(* Logix 5000 project; controller SX_V040001_C001 vendor 1 type 14 code 77 rev 16.22; software revision 16.04; part 5 of 35 *)
(* tags used below, declared in another part *)
   ALARM_BITS : INT[10];
   ALL_KINDS : INT[90];
   Basic : INT;
   EMPTYING : INT[18];
   G_AInput : DINT[8];
   G_DInput : DINT[3];
   G_DOutput : DINT[3];
   loading : INT[19];
   m_alarm_exist : BOOL;
   m_notstop : BOOL;
   METERING : INT[44];
   PARAMETER : INT[501];
   T_AIR_PRESSURE : TIMER;
   T_BEARING_LUBR : TIMER;
   T_CHOCO_PRESSURE : TIMER;
   T_DELAY_BROKEN_AI_0 : TIMER;
   T_DELAY_BROKEN_AI_1 : TIMER;
   T_DELAY_BROKEN_AI_2 : TIMER;
   T_DELAY_BROKEN_AI_3 : TIMER;
   T_DELAY_BROKEN_AI_4 : TIMER;
   T_DELAY_BROKEN_AI_5 : TIMER;
   T_DELAY_BROKEN_AI_6 : TIMER;
   T_DELAY_BROKEN_AI_7 : TIMER;
   T_INLETT_VALVE : TIMER;
   T_STUFFINGBOX_LUBR : TIMER;
   TEMP : INT[14];
   Z30 : COUNTER;
   Z31 : COUNTER;
   Z33 : COUNTER;
   Z34 : COUNTER;
   Z35 : COUNTER;
   Z36 : COUNTER;
   Z37 : COUNTER;
   Z38 : COUNTER;
   Z39 : COUNTER;
   Z40 : COUNTER;
   Z41 : COUNTER;
(* MainProgram, continued *)

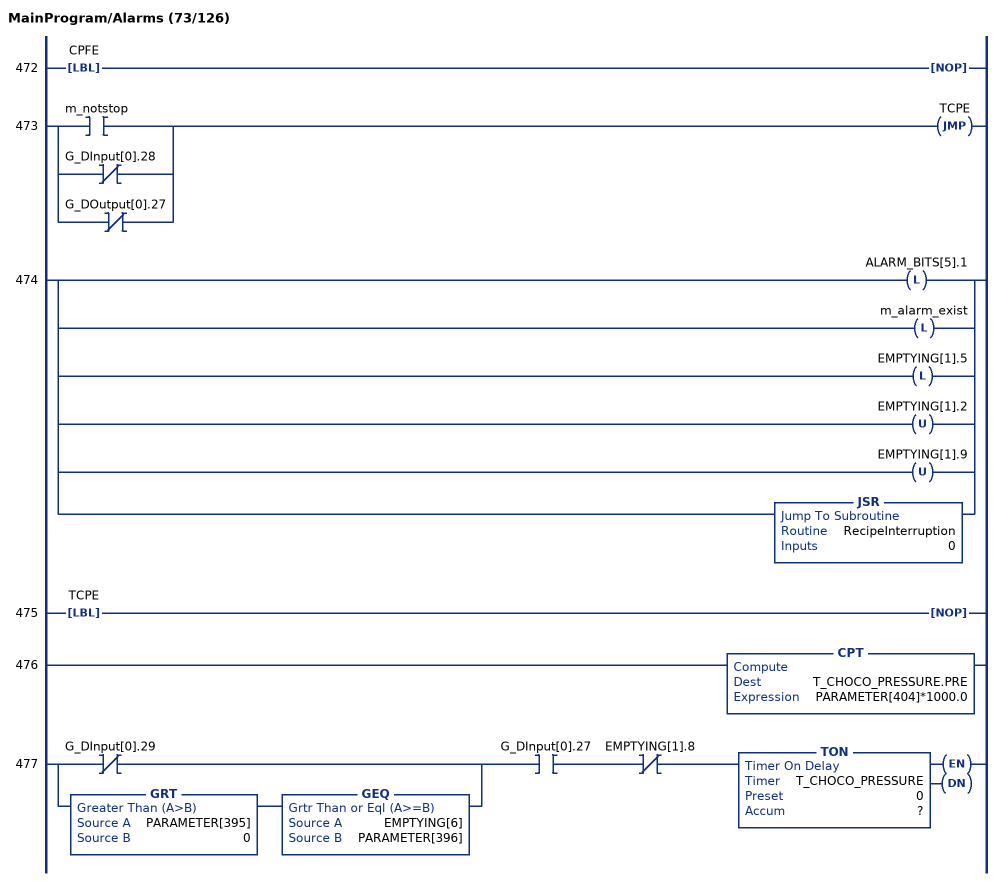
   [picture p94: MainProgram/Alarms rungs 472-477]
   472: LBL(CPFE)NOP();
   473: [XIC(m_notstop) ,XIO(G_DInput[0].28) ,XIO(G_DOutput[0].27) ]JMP(TCPE);
   474: [OTL(ALARM_BITS[5].1) ,OTL(m_alarm_exist) ,OTL(EMPTYING[1].5) ,OTU(EMPTYING[1].2) ,OTU(EMPTYING[1].9) ,JSR(RecipeInterruption,0) ];
   475: LBL(TCPE)NOP();
   476: CPT(T_CHOCO_PRESSURE.PRE,PARAMETER[404]*1000.0);
   477: [XIO(G_DInput[0].29) ,GRT(PARAMETER[395],0) GEQ(EMPTYING[6],PARAMETER[396]) ]XIC(G_DInput[0].27)XIO(EMPTYING[1].8)TON(T_CHOCO_PRESSURE,?,?);
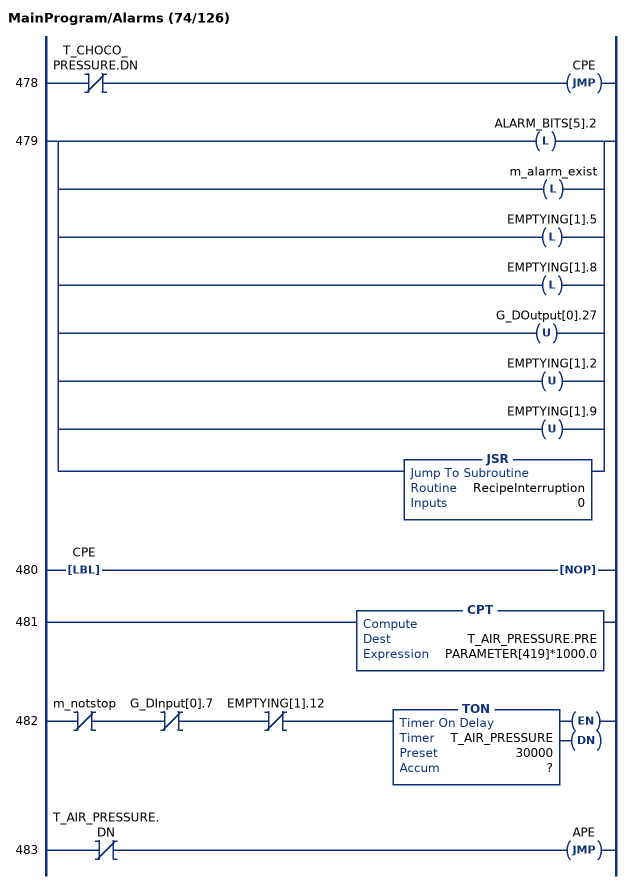
   478: XIO(T_CHOCO_PRESSURE.DN)JMP(CPE);
   479: [OTL(ALARM_BITS[5].2) ,OTL(m_alarm_exist) ,OTL(EMPTYING[1].5) ,OTL(EMPTYING[1].8) ,OTU(G_DOutput[0].27) ,OTU(EMPTYING[1].2) ,OTU(EMPTYING[1].9) ,JSR(RecipeInterruption,0) ];
   480: LBL(CPE)NOP();
   481: CPT(T_AIR_PRESSURE.PRE,PARAMETER[419]*1000.0);
   482: XIO(m_notstop)XIO(G_DInput[0].7)XIO(EMPTYING[1].12)TON(T_AIR_PRESSURE,?,?);
   483: XIO(T_AIR_PRESSURE.DN)JMP(APE);
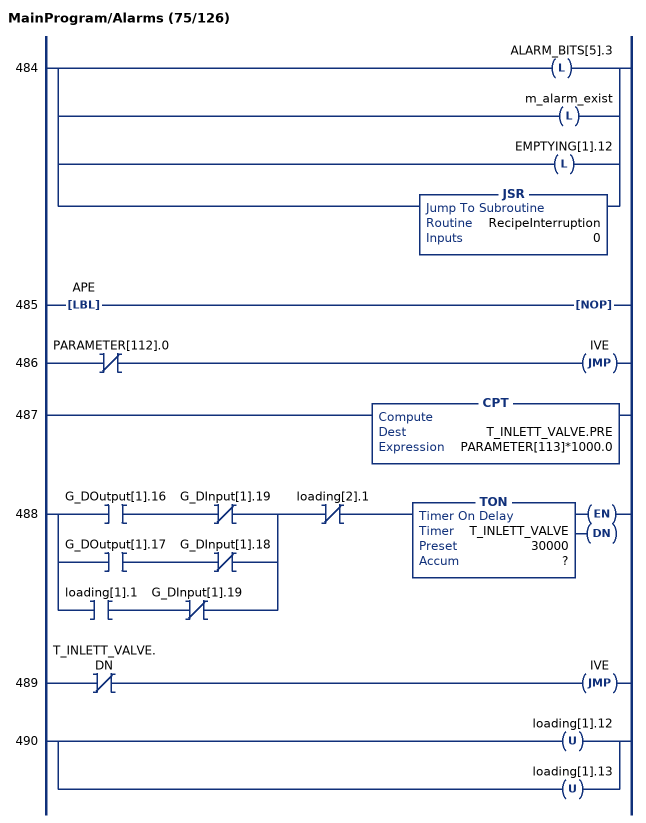
   484: [OTL(ALARM_BITS[5].3) ,OTL(m_alarm_exist) ,OTL(EMPTYING[1].12) ,JSR(RecipeInterruption,0) ];
   485: LBL(APE)NOP();
   486: XIO(PARAMETER[112].0)JMP(IVE);
   487: CPT(T_INLETT_VALVE.PRE,PARAMETER[113]*1000.0);
   488: [XIC(G_DOutput[1].16) XIO(G_DInput[1].19) ,XIC(G_DOutput[1].17) XIO(G_DInput[1].18) ,XIC(loading[1].1) XIO(G_DInput[1].19) ]XIO(loading[2].1)TON(T_INLETT_VALVE,?,?);
   489: XIO(T_INLETT_VALVE.DN)JMP(IVE);
   490: [OTU(loading[1].12) ,OTU(loading[1].13) ];
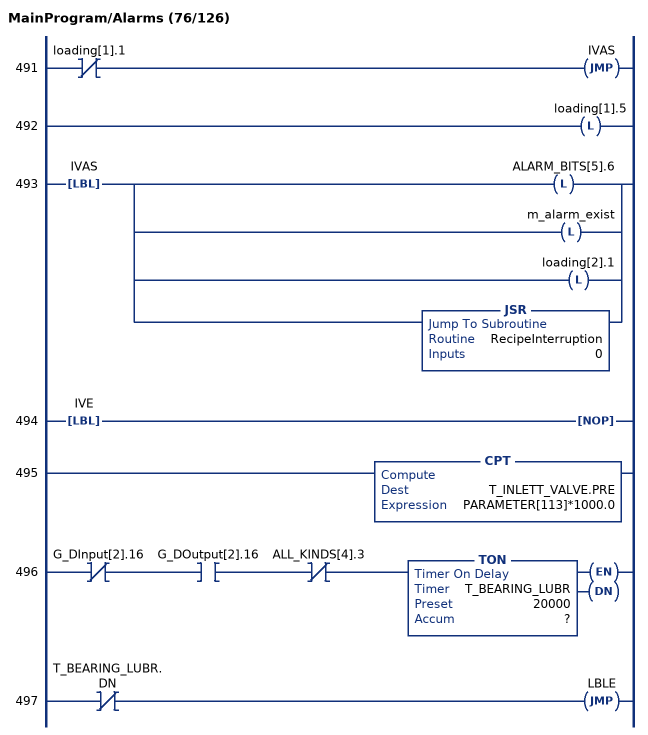
   491: XIO(loading[1].1)JMP(IVAS);
   492: OTL(loading[1].5);
   493: LBL(IVAS)[OTL(ALARM_BITS[5].6) ,OTL(m_alarm_exist) ,OTL(loading[2].1) ,JSR(RecipeInterruption,0) ];
   494: LBL(IVE)NOP();
   495: CPT(T_INLETT_VALVE.PRE,PARAMETER[113]*1000.0);
   496: XIO(G_DInput[2].16)XIC(G_DOutput[2].16)XIO(ALL_KINDS[4].3)TON(T_BEARING_LUBR,?,?);
   497: XIO(T_BEARING_LUBR.DN)JMP(LBLE);
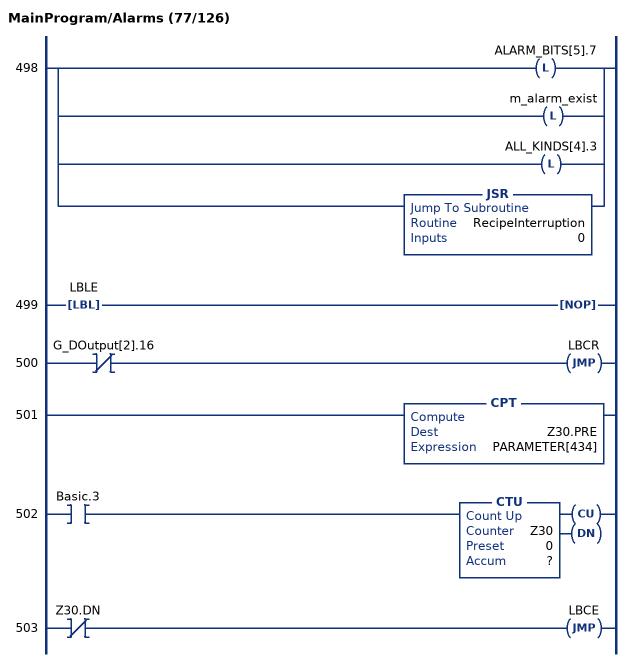
   498: [OTL(ALARM_BITS[5].7) ,OTL(m_alarm_exist) ,OTL(ALL_KINDS[4].3) ,JSR(RecipeInterruption,0) ];
   499: LBL(LBLE)NOP();
   500: XIO(G_DOutput[2].16)JMP(LBCR);
   501: CPT(Z30.PRE,PARAMETER[434]);
   502: XIC(Basic.3)CTU(Z30,?,?);
   503: XIO(Z30.DN)JMP(LBCE);
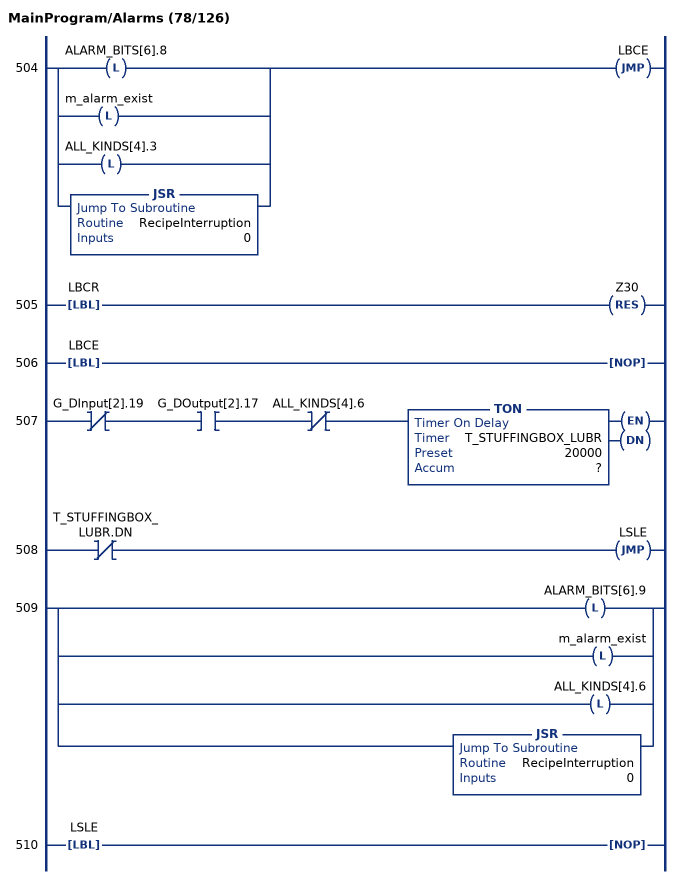
   504: [OTL(ALARM_BITS[6].8) ,OTL(m_alarm_exist) ,OTL(ALL_KINDS[4].3) ,JSR(RecipeInterruption,0) ]JMP(LBCE);
   505: LBL(LBCR)RES(Z30);
   506: LBL(LBCE)NOP();
   507: XIO(G_DInput[2].19)XIC(G_DOutput[2].17)XIO(ALL_KINDS[4].6)TON(T_STUFFINGBOX_LUBR,?,?);
   508: XIO(T_STUFFINGBOX_LUBR.DN)JMP(LSLE);
   509: [OTL(ALARM_BITS[6].9) ,OTL(m_alarm_exist) ,OTL(ALL_KINDS[4].6) ,JSR(RecipeInterruption,0) ];
   510: LBL(LSLE)NOP();
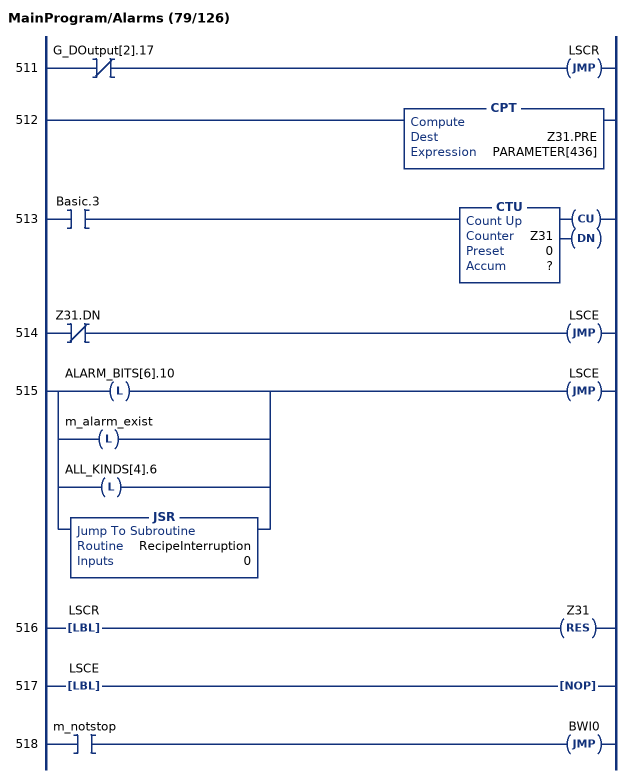
   511: XIO(G_DOutput[2].17)JMP(LSCR);
   512: CPT(Z31.PRE,PARAMETER[436]);
   513: XIC(Basic.3)CTU(Z31,?,?);
   514: XIO(Z31.DN)JMP(LSCE);
   515: [OTL(ALARM_BITS[6].10) ,OTL(m_alarm_exist) ,OTL(ALL_KINDS[4].6) ,JSR(RecipeInterruption,0) ]JMP(LSCE);
   516: LBL(LSCR)RES(Z31);
   517: LBL(LSCE)NOP();
   518: XIC(m_notstop)JMP(BWI0);
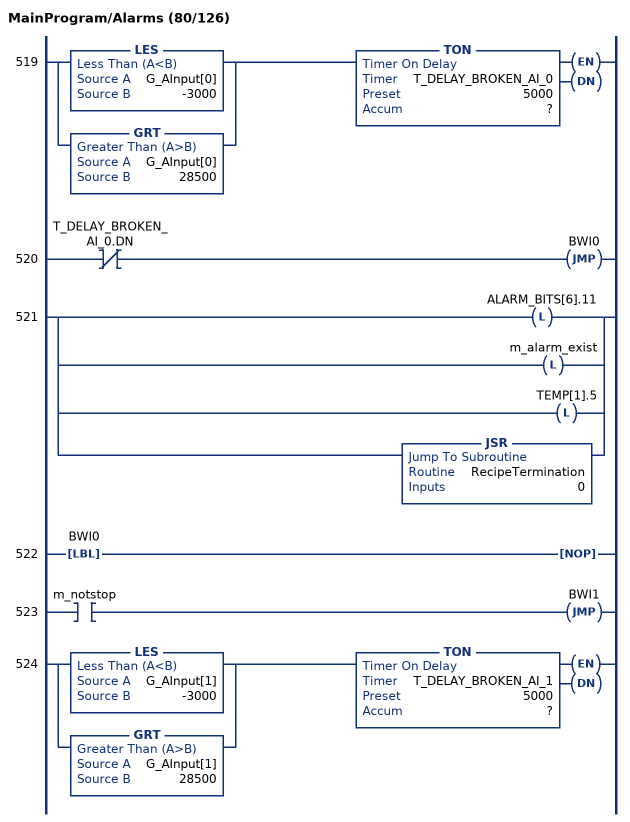
   519: [LES(G_AInput[0],-3000) ,GRT(G_AInput[0],28500) ]TON(T_DELAY_BROKEN_AI_0,?,?);
   520: XIO(T_DELAY_BROKEN_AI_0.DN)JMP(BWI0);
   521: [OTL(ALARM_BITS[6].11) ,OTL(m_alarm_exist) ,OTL(TEMP[1].5) ,JSR(RecipeTermination,0) ];
   522: LBL(BWI0)NOP();
   523: XIC(m_notstop)JMP(BWI1);
   524: [LES(G_AInput[1],-3000) ,GRT(G_AInput[1],28500) ]TON(T_DELAY_BROKEN_AI_1,?,?);
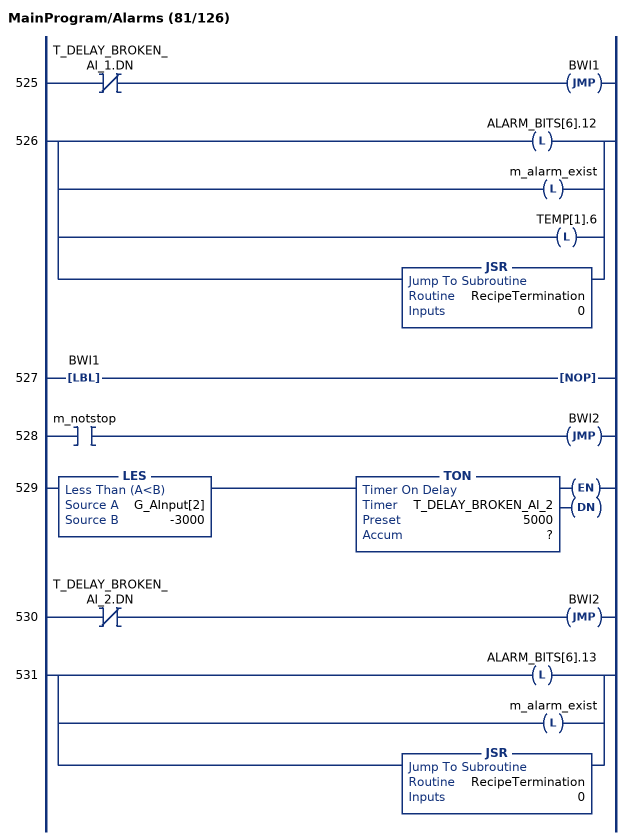
   525: XIO(T_DELAY_BROKEN_AI_1.DN)JMP(BWI1);
   526: [OTL(ALARM_BITS[6].12) ,OTL(m_alarm_exist) ,OTL(TEMP[1].6) ,JSR(RecipeTermination,0) ];
   527: LBL(BWI1)NOP();
   528: XIC(m_notstop)JMP(BWI2);
   529: LES(G_AInput[2],-3000)TON(T_DELAY_BROKEN_AI_2,?,?);
   530: XIO(T_DELAY_BROKEN_AI_2.DN)JMP(BWI2);
   531: [OTL(ALARM_BITS[6].13) ,OTL(m_alarm_exist) ,JSR(RecipeTermination,0) ];
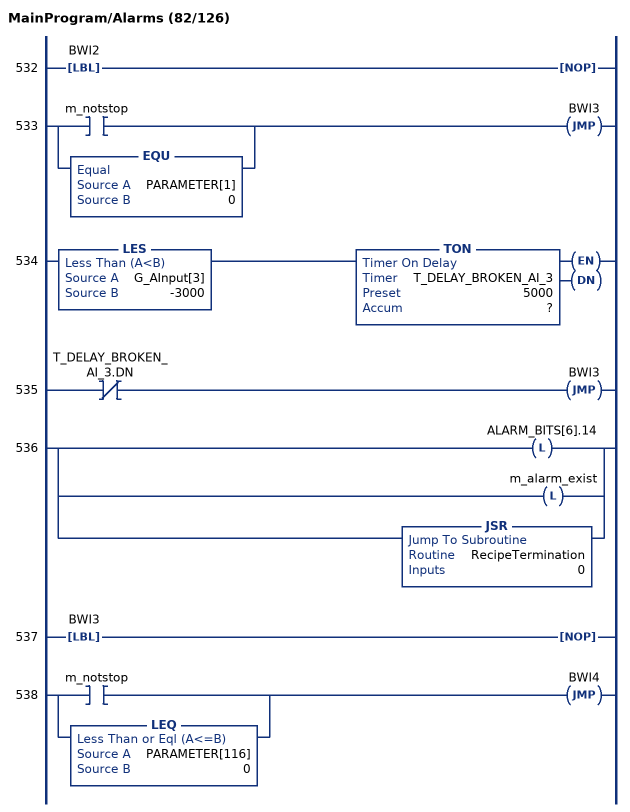
   532: LBL(BWI2)NOP();
   533: [XIC(m_notstop) ,EQU(PARAMETER[1],0) ]JMP(BWI3);
   534: LES(G_AInput[3],-3000)TON(T_DELAY_BROKEN_AI_3,?,?);
   535: XIO(T_DELAY_BROKEN_AI_3.DN)JMP(BWI3);
   536: [OTL(ALARM_BITS[6].14) ,OTL(m_alarm_exist) ,JSR(RecipeTermination,0) ];
   537: LBL(BWI3)NOP();
   538: [XIC(m_notstop) ,LEQ(PARAMETER[116],0) ]JMP(BWI4);
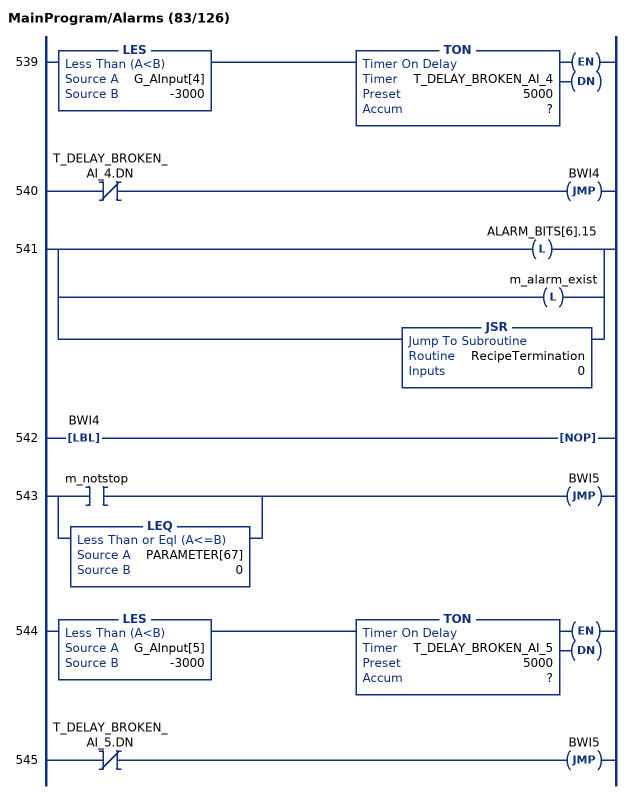
   539: LES(G_AInput[4],-3000)TON(T_DELAY_BROKEN_AI_4,?,?);
   540: XIO(T_DELAY_BROKEN_AI_4.DN)JMP(BWI4);
   541: [OTL(ALARM_BITS[6].15) ,OTL(m_alarm_exist) ,JSR(RecipeTermination,0) ];
   542: LBL(BWI4)NOP();
   543: [XIC(m_notstop) ,LEQ(PARAMETER[67],0) ]JMP(BWI5);
   544: LES(G_AInput[5],-3000)TON(T_DELAY_BROKEN_AI_5,?,?);
   545: XIO(T_DELAY_BROKEN_AI_5.DN)JMP(BWI5);
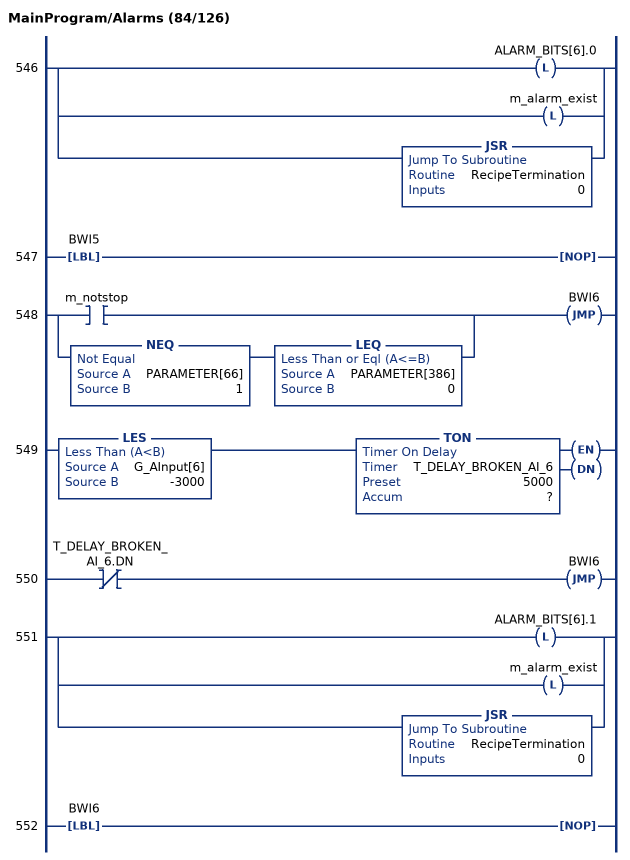
   546: [OTL(ALARM_BITS[6].0) ,OTL(m_alarm_exist) ,JSR(RecipeTermination,0) ];
   547: LBL(BWI5)NOP();
   548: [XIC(m_notstop) ,NEQ(PARAMETER[66],1) LEQ(PARAMETER[386],0) ]JMP(BWI6);
   549: LES(G_AInput[6],-3000)TON(T_DELAY_BROKEN_AI_6,?,?);
   550: XIO(T_DELAY_BROKEN_AI_6.DN)JMP(BWI6);
   551: [OTL(ALARM_BITS[6].1) ,OTL(m_alarm_exist) ,JSR(RecipeTermination,0) ];
   552: LBL(BWI6)NOP();
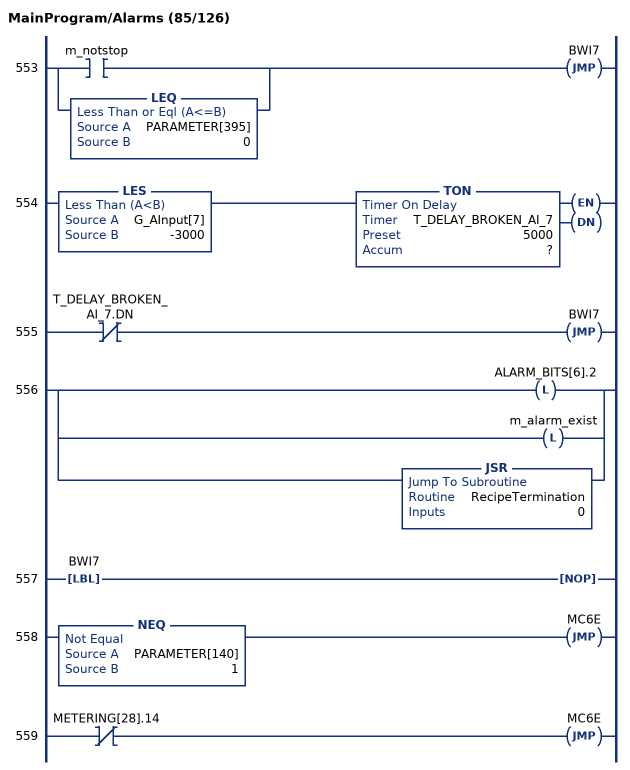
   553: [XIC(m_notstop) ,LEQ(PARAMETER[395],0) ]JMP(BWI7);
   554: LES(G_AInput[7],-3000)TON(T_DELAY_BROKEN_AI_7,?,?);
   555: XIO(T_DELAY_BROKEN_AI_7.DN)JMP(BWI7);
   556: [OTL(ALARM_BITS[6].2) ,OTL(m_alarm_exist) ,JSR(RecipeTermination,0) ];
   557: LBL(BWI7)NOP();
   558: NEQ(PARAMETER[140],1)JMP(MC6E);
   559: XIO(METERING[28].14)JMP(MC6E);
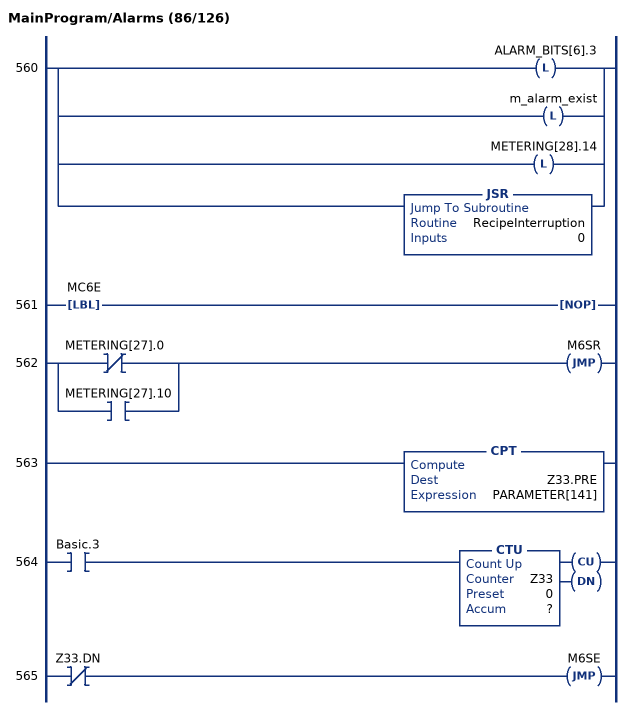
   560: [OTL(ALARM_BITS[6].3) ,OTL(m_alarm_exist) ,OTL(METERING[28].14) ,JSR(RecipeInterruption,0) ];
   561: LBL(MC6E)NOP();
   562: [XIO(METERING[27].0) ,XIC(METERING[27].10) ]JMP(M6SR);
   563: CPT(Z33.PRE,PARAMETER[141]);
   564: XIC(Basic.3)CTU(Z33,?,?);
   565: XIO(Z33.DN)JMP(M6SE);
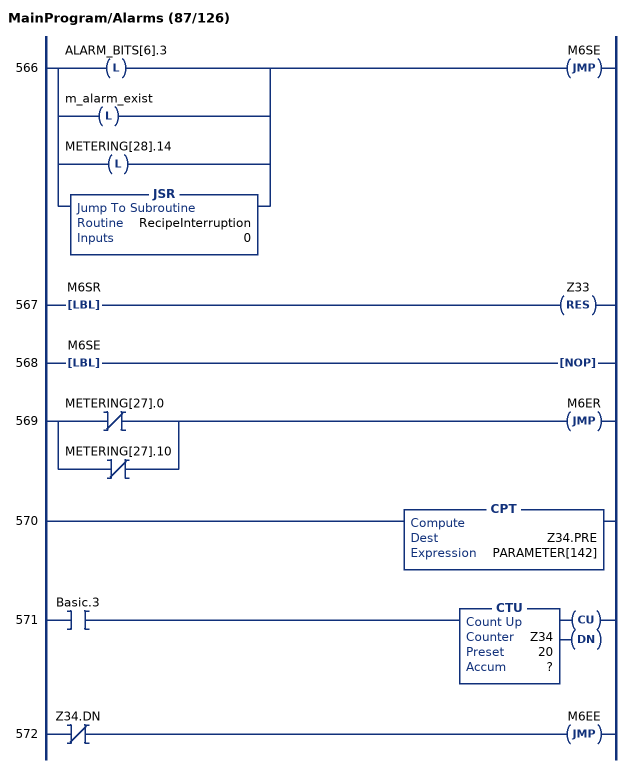
   566: [OTL(ALARM_BITS[6].3) ,OTL(m_alarm_exist) ,OTL(METERING[28].14) ,JSR(RecipeInterruption,0) ]JMP(M6SE);
   567: LBL(M6SR)RES(Z33);
   568: LBL(M6SE)NOP();
   569: [XIO(METERING[27].0) ,XIO(METERING[27].10) ]JMP(M6ER);
   570: CPT(Z34.PRE,PARAMETER[142]);
   571: XIC(Basic.3)CTU(Z34,?,?);
   572: XIO(Z34.DN)JMP(M6EE);
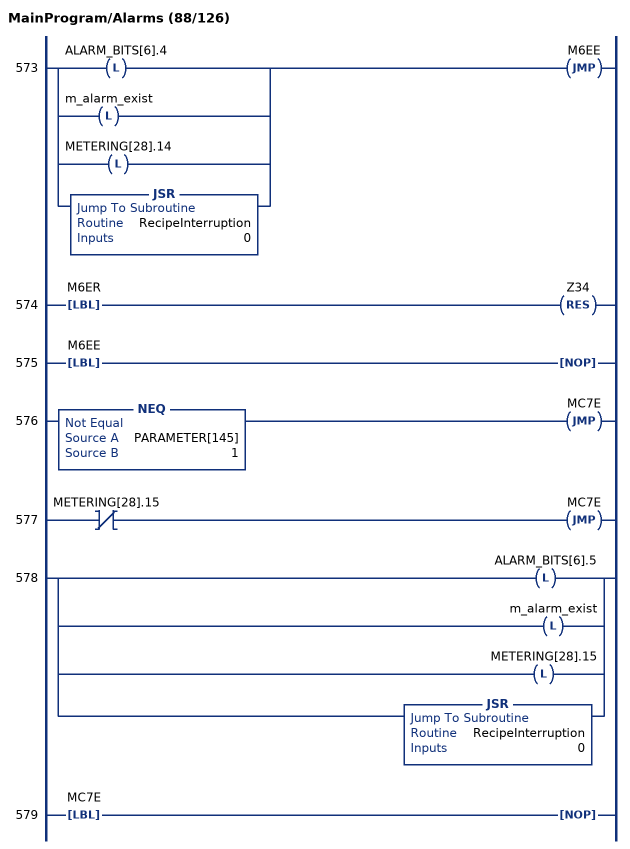
   573: [OTL(ALARM_BITS[6].4) ,OTL(m_alarm_exist) ,OTL(METERING[28].14) ,JSR(RecipeInterruption,0) ]JMP(M6EE);
   574: LBL(M6ER)RES(Z34);
   575: LBL(M6EE)NOP();
   576: NEQ(PARAMETER[145],1)JMP(MC7E);
   577: XIO(METERING[28].15)JMP(MC7E);
   578: [OTL(ALARM_BITS[6].5) ,OTL(m_alarm_exist) ,OTL(METERING[28].15) ,JSR(RecipeInterruption,0) ];
   579: LBL(MC7E)NOP();
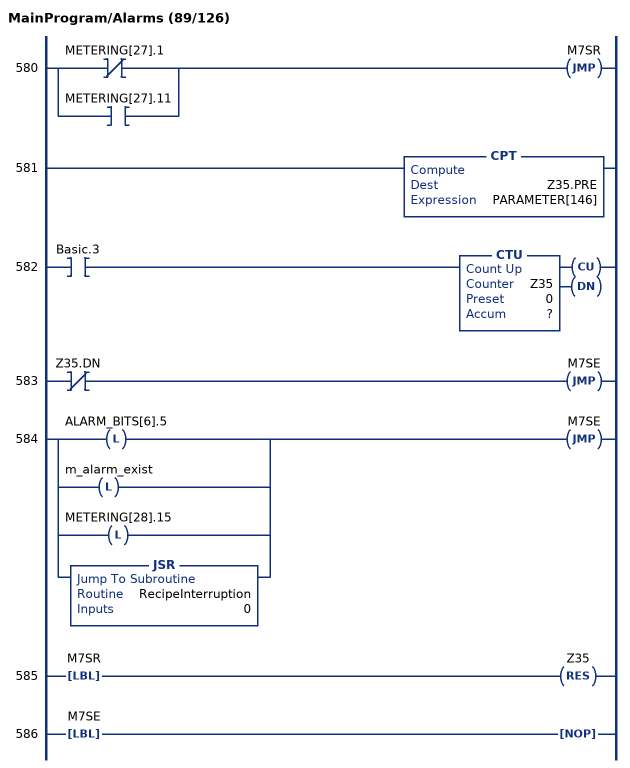
   580: [XIO(METERING[27].1) ,XIC(METERING[27].11) ]JMP(M7SR);
   581: CPT(Z35.PRE,PARAMETER[146]);
   582: XIC(Basic.3)CTU(Z35,?,?);
   583: XIO(Z35.DN)JMP(M7SE);
   584: [OTL(ALARM_BITS[6].5) ,OTL(m_alarm_exist) ,OTL(METERING[28].15) ,JSR(RecipeInterruption,0) ]JMP(M7SE);
   585: LBL(M7SR)RES(Z35);
   586: LBL(M7SE)NOP();
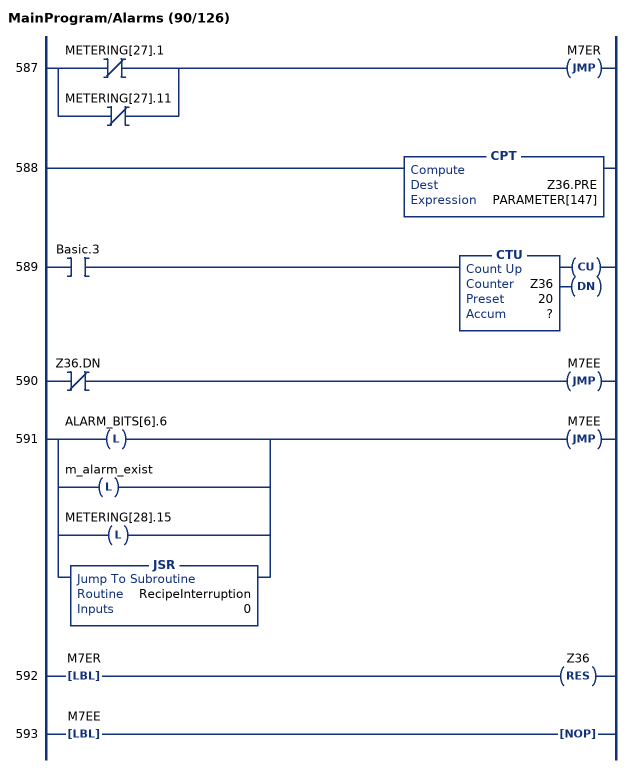
   587: [XIO(METERING[27].1) ,XIO(METERING[27].11) ]JMP(M7ER);
   588: CPT(Z36.PRE,PARAMETER[147]);
   589: XIC(Basic.3)CTU(Z36,?,?);
   590: XIO(Z36.DN)JMP(M7EE);
   591: [OTL(ALARM_BITS[6].6) ,OTL(m_alarm_exist) ,OTL(METERING[28].15) ,JSR(RecipeInterruption,0) ]JMP(M7EE);
   592: LBL(M7ER)RES(Z36);
   593: LBL(M7EE)NOP();
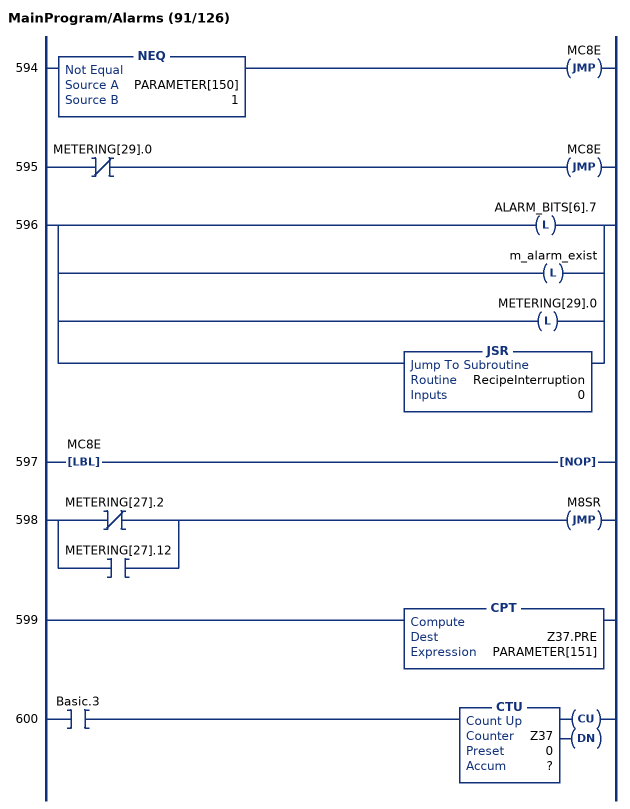
   594: NEQ(PARAMETER[150],1)JMP(MC8E);
   595: XIO(METERING[29].0)JMP(MC8E);
   596: [OTL(ALARM_BITS[6].7) ,OTL(m_alarm_exist) ,OTL(METERING[29].0) ,JSR(RecipeInterruption,0) ];
   597: LBL(MC8E)NOP();
   598: [XIO(METERING[27].2) ,XIC(METERING[27].12) ]JMP(M8SR);
   599: CPT(Z37.PRE,PARAMETER[151]);
   600: XIC(Basic.3)CTU(Z37,?,?);
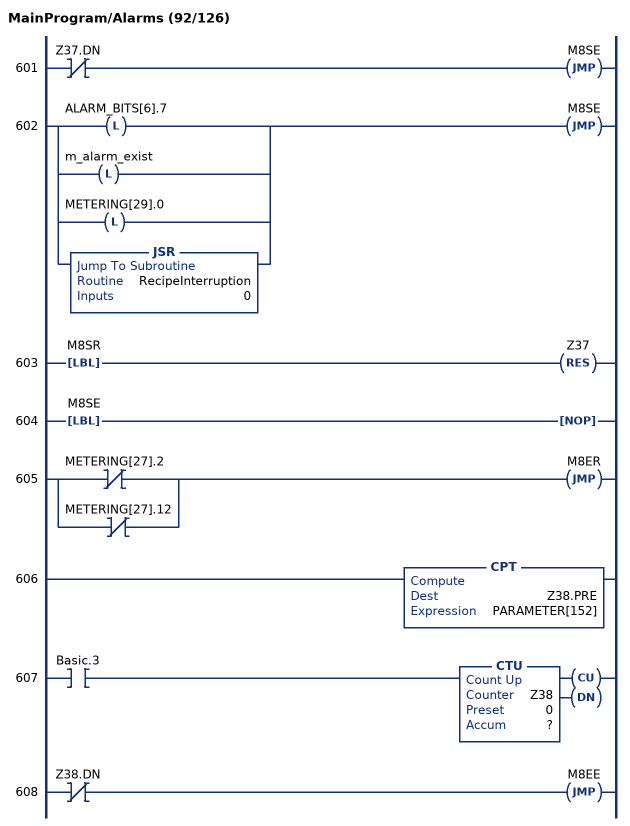
   601: XIO(Z37.DN)JMP(M8SE);
   602: [OTL(ALARM_BITS[6].7) ,OTL(m_alarm_exist) ,OTL(METERING[29].0) ,JSR(RecipeInterruption,0) ]JMP(M8SE);
   603: LBL(M8SR)RES(Z37);
   604: LBL(M8SE)NOP();
   605: [XIO(METERING[27].2) ,XIO(METERING[27].12) ]JMP(M8ER);
   606: CPT(Z38.PRE,PARAMETER[152]);
   607: XIC(Basic.3)CTU(Z38,?,?);
   608: XIO(Z38.DN)JMP(M8EE);
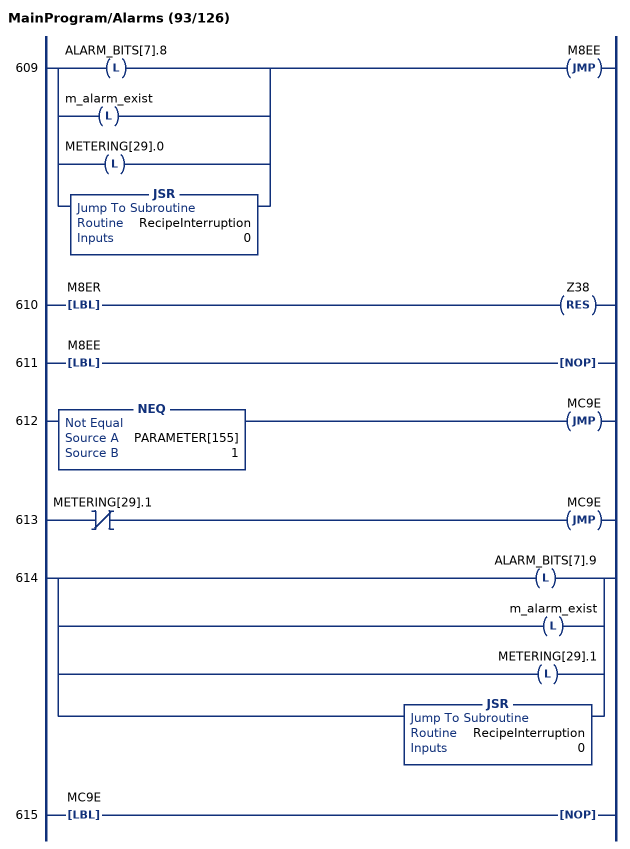
   609: [OTL(ALARM_BITS[7].8) ,OTL(m_alarm_exist) ,OTL(METERING[29].0) ,JSR(RecipeInterruption,0) ]JMP(M8EE);
   610: LBL(M8ER)RES(Z38);
   611: LBL(M8EE)NOP();
   612: NEQ(PARAMETER[155],1)JMP(MC9E);
   613: XIO(METERING[29].1)JMP(MC9E);
   614: [OTL(ALARM_BITS[7].9) ,OTL(m_alarm_exist) ,OTL(METERING[29].1) ,JSR(RecipeInterruption,0) ];
   615: LBL(MC9E)NOP();
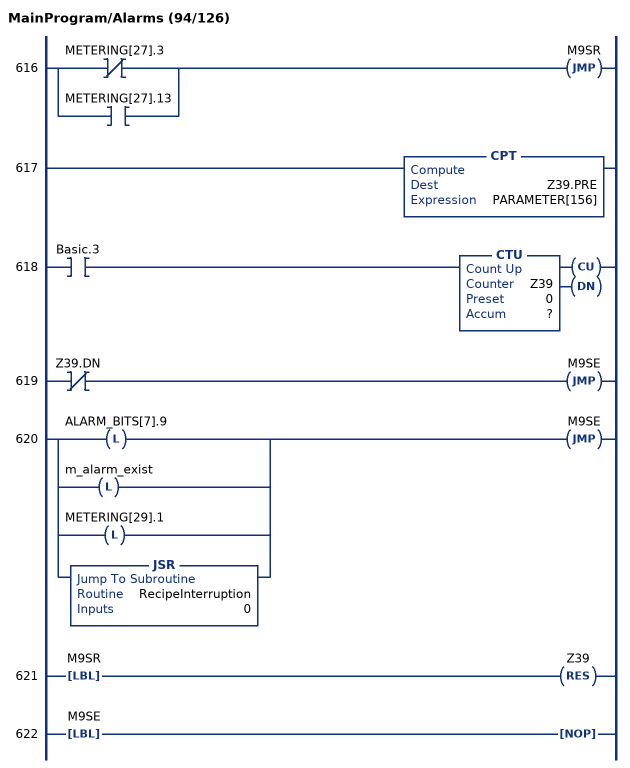
   616: [XIO(METERING[27].3) ,XIC(METERING[27].13) ]JMP(M9SR);
   617: CPT(Z39.PRE,PARAMETER[156]);
   618: XIC(Basic.3)CTU(Z39,?,?);
   619: XIO(Z39.DN)JMP(M9SE);
   620: [OTL(ALARM_BITS[7].9) ,OTL(m_alarm_exist) ,OTL(METERING[29].1) ,JSR(RecipeInterruption,0) ]JMP(M9SE);
   621: LBL(M9SR)RES(Z39);
   622: LBL(M9SE)NOP();
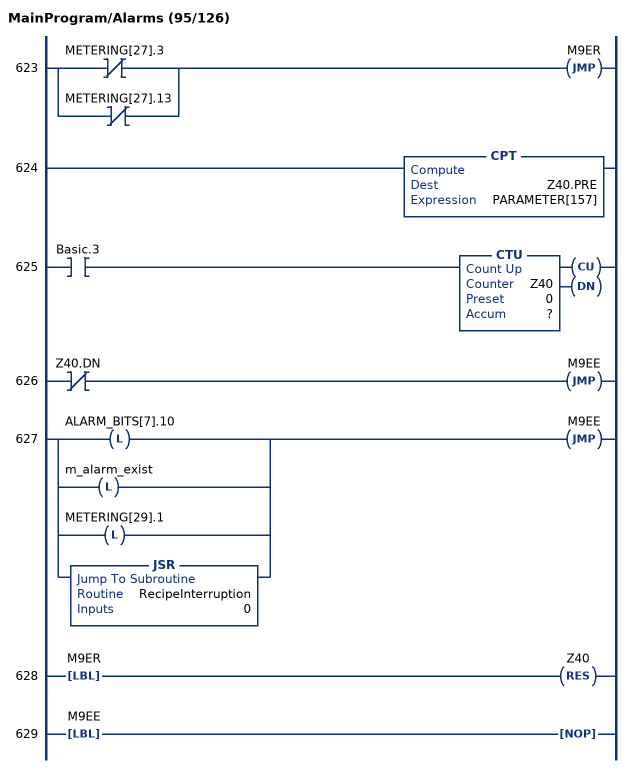
   623: [XIO(METERING[27].3) ,XIO(METERING[27].13) ]JMP(M9ER);
   624: CPT(Z40.PRE,PARAMETER[157]);
   625: XIC(Basic.3)CTU(Z40,?,?);
   626: XIO(Z40.DN)JMP(M9EE);
   627: [OTL(ALARM_BITS[7].10) ,OTL(m_alarm_exist) ,OTL(METERING[29].1) ,JSR(RecipeInterruption,0) ]JMP(M9EE);
   628: LBL(M9ER)RES(Z40);
   629: LBL(M9EE)NOP();
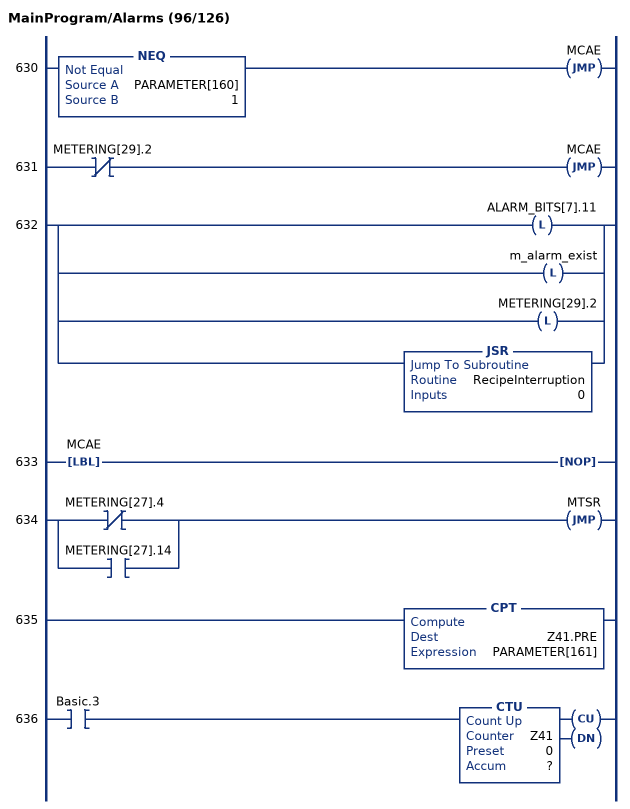
   630: NEQ(PARAMETER[160],1)JMP(MCAE);
   631: XIO(METERING[29].2)JMP(MCAE);
   632: [OTL(ALARM_BITS[7].11) ,OTL(m_alarm_exist) ,OTL(METERING[29].2) ,JSR(RecipeInterruption,0) ];
   633: LBL(MCAE)NOP();
   634: [XIO(METERING[27].4) ,XIC(METERING[27].14) ]JMP(MTSR);
   635: CPT(Z41.PRE,PARAMETER[161]);
   636: XIC(Basic.3)CTU(Z41,?,?);
